{attribute 'linkalways'} 
{attribute 'no_explicit_call' := 'This FB is a CLASS and must be accessed using methods or properties'}
{attribute 'enable_dynamic_creation'}
FUNCTION_BLOCK _ETcVnFeatureDescriptorTypeAKAZE EXTENDS EnumDatatypeBase
VAR
	localData : ETcVnFeatureDescriptorTypeAKAZE;
	activeData : REFERENCE TO ETcVnFeatureDescriptorTypeAKAZE;
	enumBaseDatatype : _DINT(localData);
END_VAR

METHOD PRIVATE AddLocalEnumeration
VAR_INPUT
	Enumeration : T_MAXSTRING;
	Value : ETcVnFeatureDescriptorTypeAKAZE;
END_VAR
AddEnumeration(Enumeration, Value);
END_METHOD

PROPERTY PUBLIC Address : PVOID
GET
Address := ADR(activeData);
END_GET
END_PROPERTY

METHOD PUBLIC ClearReference
VAR_INPUT
END_VAR
activeData REF= localData;
SetBaseDatatypeReference();
END_METHOD

METHOD PUBLIC Clone : I_Datatype
VAR
    pClone : POINTER TO _ETcVnFeatureDescriptorTypeAKAZE;
END_VAR
pClone := __NEW(_ETcVnFeatureDescriptorTypeAKAZE(InitialValue := Value));
Clone := pClone^;
END_METHOD

METHOD FB_init : BOOL
VAR_INPUT
	bInitRetains : BOOL; // if TRUE, the retain variables are initialized (warm start / cold start)
	bInCopyCode : BOOL;  // if TRUE, the instance afterwards gets moved into the copy code (online change)
	InitialValue : ETcVnFeatureDescriptorTypeAKAZE;
END_VAR
localData := InitialValue;
AddBaseDatatype(enumBaseDatatype);
ClearReference();

AddLocalEnumeration('TCVN_FDT_AKAZE_KAZE_UPRIGHT', ETcVnFeatureDescriptorTypeAKAZE.TCVN_FDT_AKAZE_KAZE_UPRIGHT);
AddLocalEnumeration('TCVN_FDT_AKAZE_KAZE', ETcVnFeatureDescriptorTypeAKAZE.TCVN_FDT_AKAZE_KAZE);
AddLocalEnumeration('TCVN_FDT_AKAZE_MLDB_UPRIGHT', ETcVnFeatureDescriptorTypeAKAZE.TCVN_FDT_AKAZE_MLDB_UPRIGHT);
AddLocalEnumeration('TCVN_FDT_AKAZE_MLDB', ETcVnFeatureDescriptorTypeAKAZE.TCVN_FDT_AKAZE_MLDB);
END_METHOD

PROPERTY PUBLIC Identifier : T_MAXSTRING
GET
Identifier := 'ETcVnFeatureDescriptorTypeAKAZE';
END_GET
END_PROPERTY

METHOD IsEnumeratorValueEqual : BOOL
VAR_INPUT
	Enumerator : I_KeyValueForwardEnumerator;
END_VAR
VAR
	storedValue : ETcVnFeatureDescriptorTypeAKAZE;
END_VAR
IF NOT Enumerator.TryGet(storedValue) THEN
	RETURN;
END_IF

IsEnumeratorValueEqual := storedValue = activeData;
END_METHOD

METHOD PUBLIC MakeReferenceTo
VAR_INPUT
	ReferenceTarget : REFERENCE TO ETcVnFeatureDescriptorTypeAKAZE;
END_VAR
activeData REF= ReferenceTarget;
SetBaseDatatypeReference();
END_METHOD

METHOD PROTECTED SetBaseDatatypeReference
VAR_INPUT
END_VAR
enumBaseDatatype.MakeReferenceTo(activeData);
END_METHOD

PROPERTY PUBLIC Size : UDINT
GET
Size := SIZEOF(activeData);
END_GET
END_PROPERTY

METHOD TryMakeReferenceTo : BOOL
VAR_INPUT
	Target : I_Datatype;
END_VAR
VAR
	targetAsEnum : I_EnumDatatype;
	pTargetData : POINTER TO ETcVnFeatureDescriptorTypeAKAZE;
END_VAR
IF NOT Target.TryResolveAsEnumDatatype(targetAsEnum) THEN
	RETURN;
END_IF

IF targetAsEnum.Identifier <> Identifier THEN
	RETURN;
END_IF

pTargetData := Target.Address;
activeData REF= pTargetData^;
SetBaseDatatypeReference();
TryMakeReferenceTo := TRUE;
END_METHOD

PROPERTY PUBLIC Value : ETcVnFeatureDescriptorTypeAKAZE
GET
Value := activeData;
END_GET
SET
activeData := Value;
END_SET
END_PROPERTY

END_FUNCTION_BLOCK

(* stored: Version 1.1.0.1, ProductVersion 3.1.4024.13
   POU _ETcVnFeatureDescriptorTypeAKAZE: Id {ce025e58-dbf3-0bca-32f1-825c1f4c9c26}, SpecialFunc None
   Folder Core: Id {df90256e-be2c-07b4-1176-ca7b7d835f25}
   Folder Protected: Id {1b39214c-64a6-039f-03e6-1c17c904f920}
   Folder Customize: Id {40879bd5-7ff4-03ba-2262-bae1b00e3d82}
   Folder Constructor: Id {58c13be2-f72d-066d-1125-a547e14edc1d}
   Folder Private: Id {6d712862-14a8-05d4-11af-0bce6a7ca7ec}
   Folder Protected: Id {5f4a540e-54c0-0bd6-01c9-9273aca4681e}
   Method AddLocalEnumeration: Id {87a5abd9-7411-0397-24fd-346a740f3478}
   Property Address: Id {a74787ca-4e9b-008a-074a-6ad900dde27d}
   Get Get: Id {0ba369d7-a5f4-0da4-1ee7-a1f15460ae17}
   Method ClearReference: Id {313ccaca-960b-0465-2b22-13fe15b51ee3}
   Method Clone: Id {ef0a1dab-8f3a-034c-1d03-c3d2b0796a15}
   Method FB_init: Id {9ed9d422-77e4-004c-3f0c-ab17e5c4aa73}
   Property Identifier: Id {47e39a47-c9ca-00fb-23fd-52d1d0517d11}
   Get Get: Id {aeaf16c5-be95-03bf-0db8-6e78433d82cf}
   Method IsEnumeratorValueEqual: Id {f6288fb3-4033-0d58-1c1e-40337b9066e8}
   Method MakeReferenceTo: Id {d2925f24-03b1-04b8-0b7c-05d56811009d}
   Method SetBaseDatatypeReference: Id {30d4aa09-20cf-0374-2f10-c314d17c365b}
   Property Size: Id {3a90c42e-377d-0fa7-16d2-879a50f3ed95}
   Get Get: Id {f800b46b-1f0d-059b-1ef7-516dbeef4ec5}
   Method TryMakeReferenceTo: Id {d5beff18-5b49-0ae5-0ff0-7516bf2e5aa4}
   Property Value: Id {5732806c-531b-0dbd-26b3-71d9f750e2ca}
   Get Get: Id {be0742cb-9821-0e56-286c-2ada18858bdc}
   Set Set: Id {5e1637b7-c599-030b-1aa8-50676f37ea04} *)
